FUNCTION_BLOCK OnOffDeviceControl
VAR
	IN AT%I* : BOOL;
	App_OnOff: BOOL;
	digitalLamp : OnOffDevice;	
	rtIN: R_TRIG;
	rtApp_IN: R_TRIG;
END_VAR

	rtIN(CLK:= IN, Q=> );
	rtApp_IN(CLK:= App_OnOff, Q=> );
	
	IF rtIN.Q THEN
		IF digitalLamp.Status = TRUE THEN
			digitalLamp.TurnOff();
		ELSE
			digitalLamp.TurnOn();
		END_IF
	END_IF

	IF rtApp_IN.Q THEN
		IF digitalLamp.Status = TRUE THEN
			digitalLamp.TurnOff();
		ELSE
			digitalLamp.TurnOn();
		END_IF
	END_IF

PROPERTY Status : BOOL
GET
Status	:=	digitalLamp.Status;
END_GET
END_PROPERTY

END_FUNCTION_BLOCK

(* stored: Version 1.1.0.1, ProductVersion 3.1.4024.13
   POU OnOffDeviceControl: Id {2dde5df7-a714-4069-814d-cd69d8282e6a}, SpecialFunc None
   Property Status: Id {edcbe291-2848-408d-b98f-780e6bbb7735}
   Get Get: Id {90a97657-631f-43c5-b91a-c03f5e73de69} *)
